// TIA Portal V18 export
FUNCTION_BLOCK "LED_FBD"   // FB54, FBD
{ S7_Optimized_Access := 'TRUE' }
VERSION : 0.1
// stored: AutoNumber true, IsIECCheckEnabled false, IsRetainMemResEnabled false, MemoryReserve 100, SetENOAutomatically false, UDAEnableTagReadback false
   VAR_INPUT
      on : Bool;
      blink : Bool;
      t_on : Time := T#1s;
      t_off : Time := T#1s;
      ignoreTestAll : Bool;
   END_VAR
   VAR_OUTPUT
      y : Bool;
   END_VAR
   VAR_IN_OUT
      testHMI : Bool;
   END_VAR
   VAR
      blink1 { S7_SetPoint := 'True'} : "BLINKER";
      blink_st : Bool;
      tonhmi { S7_SetPoint := 'True'} : TON_TIME;
   END_VAR
BEGIN

REGION Network 1
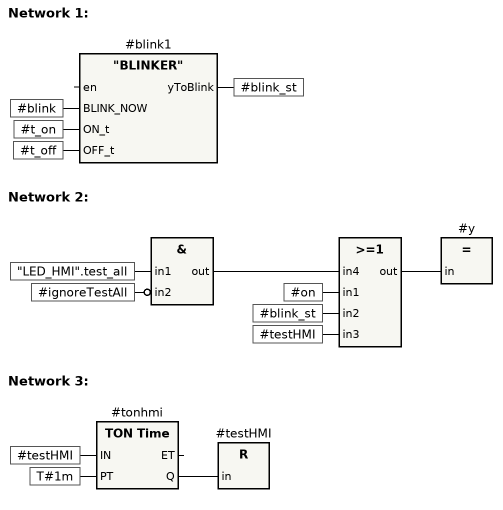
   #blink1(BLINK_NOW := #blink, ON_t := #t_on, OFF_t := #t_off, yToBlink => #blink_st);   // "BLINKER"
END_REGION

REGION Network 2
   #y := ("LED_HMI".test_all AND NOT #ignoreTestAll) OR #on OR #blink_st OR #testHMI;
END_REGION

REGION Network 3
   #tonhmi(IN := #testHMI, PT := T#1m);   // TON
   IF #tonhmi.Q THEN #testHMI := FALSE; END_IF;
END_REGION
END_FUNCTION_BLOCK
